FUNCTION_BLOCK ABSTRACT SSC_MoveWorkpiece_Base EXTENDS ControlPrimitiveBase
VAR_INPUT
END_VAR
VAR_OUTPUT
END_VAR
VAR
	m_ptrSSC: POINTER TO SmallSortingConveyor;
	
	m_step: INT := 0;
	m_TurnSwitch : BOOL;
END_VAR

SUPER^();

METHOD  Abort : BOOL
VAR_INPUT
END_VAR
m_ptrSSC^.METH_ConveyorStop();
m_ptrSSC^.METH_Switch_Retract();
Abort := TRUE;
END_METHOD

METHOD PROTECTED ABSTRACT AtTarget : BOOL
VAR_INPUT
END_VAR
END_METHOD

(* Execution logic of this Control Primitive. *)
METHOD PROTECTED ExecuteInternal : BOOL
VAR_INPUT
	i_params: ParameterSet;
END_VAR
CASE m_step OF
	0: // to target	
	IF NOT AtTarget() THEN
		m_ptrSSC^.METH_ConveyorForward();
		IF m_TurnSwitch THEN
			m_ptrSSC^.METH_Switch_Extend();
		END_IF
		m_step := 1;
	END_IF
		
	1:
	IF AtTarget() THEN
		m_ptrSSC^.METH_ConveyorStop();
		IF NOT m_TurnSwitch THEN
			m_ptrSSC^.METH_Switch_Retract();
		END_IF
		m_step := 0;
		ExecuteInternal := TRUE;
	END_IF
		
END_CASE
END_METHOD

END_FUNCTION_BLOCK

(* stored: Version 1.1.0.1
   POU SSC_MoveWorkpiece_Base: Id {43873948-1880-4c31-8462-5eebdc71c986}, SpecialFunc None
   Method Abort: Id {aa851efd-6cb5-49e3-9c58-8d0fa4675e19}
   Method AtTarget: Id {5862ac5f-4b75-49cf-a32e-243cff6373d9}
   Method ExecuteInternal: Id {f2c98800-0a51-4809-8866-e82fdec71010} *)
